TYPE U_TICKET_LIST_CTRL :
UNION
  stCtrl              : ST_LIST_CTRL;
  byCtrl    AT %Q*    : ARRAY[1..SIZEOF(ST_LIST_CTRL)] OF BYTE;
END_UNION
END_TYPE

(* stored: Version 1.1.0.1
   DUT U_TICKET_LIST_CTRL: Id {5a1aee02-c209-4656-8ace-5271f0a5b498} *)
